(* Schneider Machine Expert - Basic project PLC_Simulation, file version 2.8.0.0 *)
(* ProjectInformations: Name=New project *)

HARDWARE
  Cpu 0: TM221CE16T
  EthernetConfiguration: NetworkName=M221, IpAllocationMode=FixedAddress, IpAddress=192.168.23.101, SubnetMask=255.255.255.0
  SerialLineConfiguration: Baud=Baud19200, Parity=ParityEven, DataBits=DataBits8, StopBits=StopBits1, PhysicalMedium=PhysicalMediumRs485, TransmissionMode=TransmissionModeModbusRtu, SlaveId=1, Addressing=SlaveAddressing
  MastTask: UsePeriodScanMode=false, PeriodScan=100
  FastTask: Period=255
  CpuBehavior: StartingMode=StartAsPreviousState, AutoSaveRamOnEeprom=true, WatchdogPeriod=250

SYMBOLS  (address, symbol, comment, settings)
  %S6       SB_TB1S  "Time base of 1 s generated by an internal clock"
  %C0         [Preset=5]
  %C1         [Preset=100]

POU BlinkCoils
  (* SectionNumber=1 *)

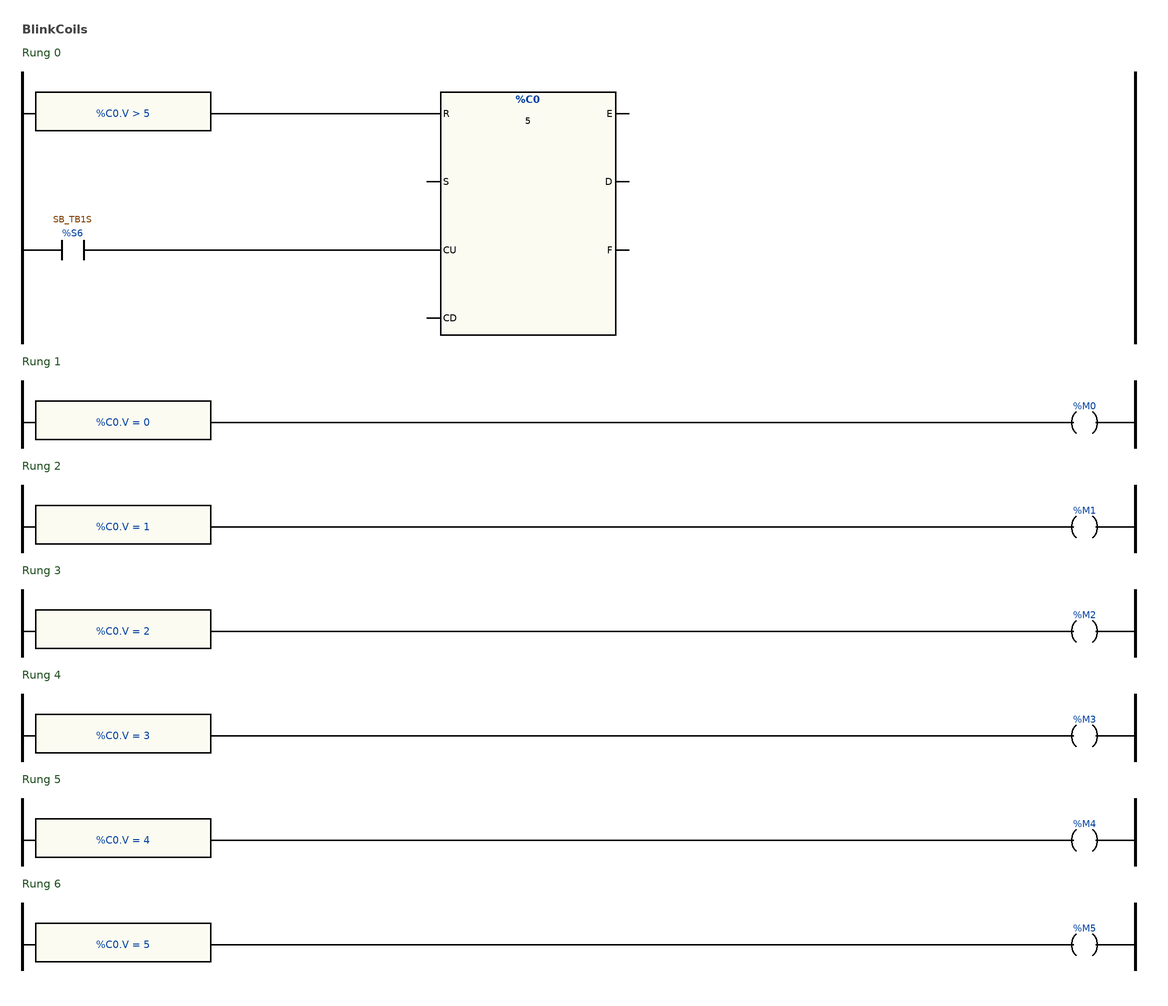

// Rung 0
  BLK %C0
  LD [ %C0.V > 5 ]
  R
  LD %S6                  (* SB_TB1S *)
  CU
  END_BLK
  // as ST:
  //   %C0(R := %C0.V > 5, CU := SB_TB1S);

// Rung 1
  LD [ %C0.V = 0 ]
  ST %M0
  // as ST:
  //   %M0 := %C0.V = 0;

// Rung 2
  LD [ %C0.V = 1 ]
  ST %M1
  // as ST:
  //   %M1 := %C0.V = 1;

// Rung 3
  LD [ %C0.V = 2 ]
  ST %M2
  // as ST:
  //   %M2 := %C0.V = 2;

// Rung 4
  LD [ %C0.V = 3 ]
  ST %M3
  // as ST:
  //   %M3 := %C0.V = 3;

// Rung 5
  LD [ %C0.V = 4 ]
  ST %M4
  // as ST:
  //   %M4 := %C0.V = 4;

// Rung 6
  LD [ %C0.V = 5 ]
  ST %M5
  // as ST:
  //   %M5 := %C0.V = 5;

POU Registers
  (* SectionNumber=2 *)

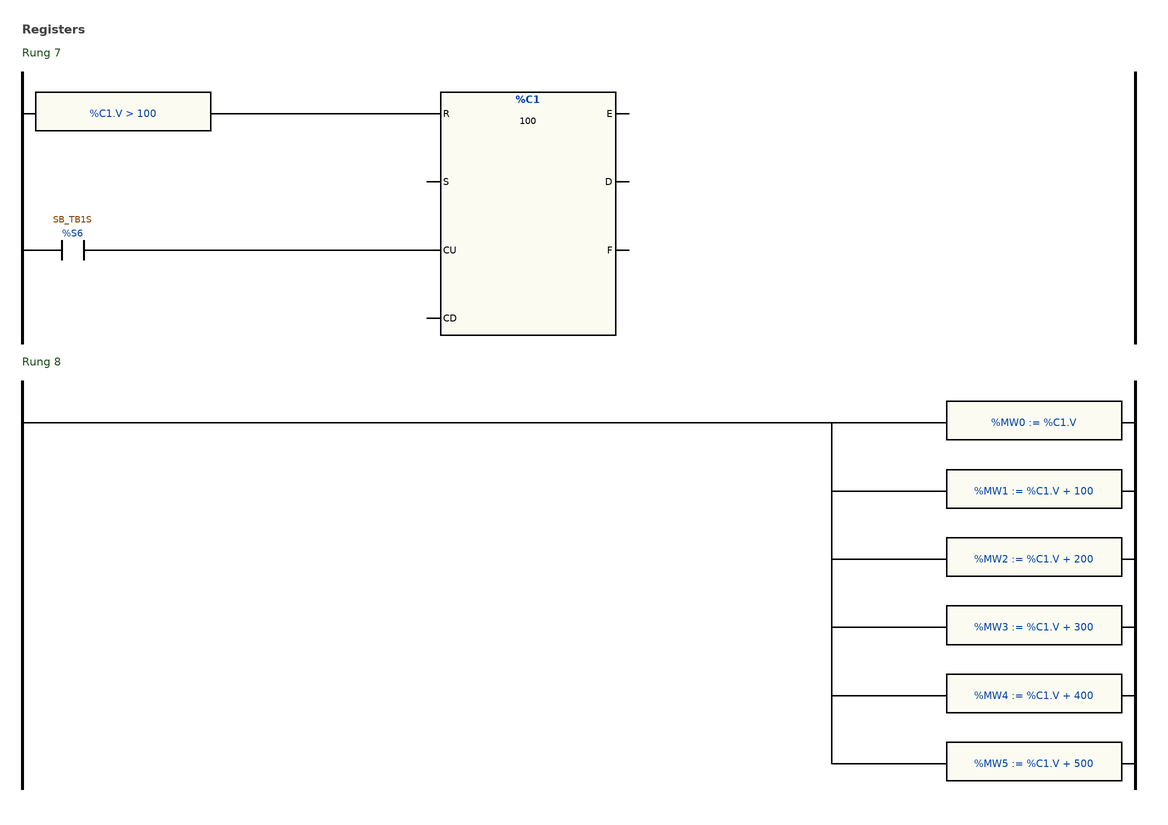

// Rung 7
  BLK %C1
  LD [ %C1.V > 100 ]
  R
  LD %S6                  (* SB_TB1S *)
  CU
  END_BLK
  // as ST:
  //   %C1(R := %C1.V > 100, CU := SB_TB1S);

// Rung 8
  LD 1
  [ %MW0 := %C1.V ]
  [ %MW1 := %C1.V + 100 ]
  [ %MW2 := %C1.V + 200 ]
  [ %MW3 := %C1.V + 300 ]
  [ %MW4 := %C1.V + 400 ]
  [ %MW5 := %C1.V + 500 ]
  // as ST:
  //   %MW0 := %C1.V;
  //   %MW1 := %C1.V + 100;
  //   %MW2 := %C1.V + 200;
  //   %MW3 := %C1.V + 300;
  //   %MW4 := %C1.V + 400;
  //   %MW5 := %C1.V + 500;
